// SIMATIC S7-200 project (STEP 7-Micro/WIN), CPU 224 CN REL 02.01

ORGANIZATION_BLOCK 主程序:OB1
TITLE=我们打算使用温度控制和数据监控确保水质处理效果。
// 具体的实现过程是这样的：系统通过模拟量输入通道接收温度传感器传来的0-20mA信号（对应0-32000的模拟值）。程序调用模拟量子程序，将信号转换为实际温度值，存储在工程值输出中。上限值设定为100.0°C，下限值设定为-50.0°C。当模拟量输入通道的值小于等于6400（对应4mA）时，工程值输出直接设为-50.0°C；当模拟量输入通道的值大于等于32000（对应20mA）时，工程值输出设为100.0°C；当模拟量输入通道的值在6400到32000之间时，通过线性插值计算出对应的温度，例如50.0°C。系统假设模拟量输入通道的值在0到32000之间，并且上限值设定大于下限值设定。
BEGIN
Network 1
LD     SM0.0
CALL   模拟量子程序:SBR3, AIW0, 100.0, -50.0, VD10
END_ORGANIZATION_BLOCK

// SBR1: protected block, not included

SUBROUTINE_BLOCK 模拟量子程序:SBR3
TITLE=
VAR_INPUT
AIW:INT;	// LW0 
HI:REAL;	// LD2 
LO:REAL;	// LD6 
END_VAR
VAR_OUTPUT
OUT:REAL;	// LD10 
END_VAR
BEGIN
Network 1 // 网络标题
// 0~20ma  对应0~32000
LD     SM0.0
ITD    #AIW:LW0, VD300
AENO
DTR    VD300, VD300
Network 2
LD     SM0.0
AR<=   VD300, 6400.0
MOVR   #LO:LD6, #OUT:LD10
Network 3
LD     SM0.0
AR>=   VD300, 32000.0
MOVR   #HI:LD2, #OUT:LD10
Network 4
LD     SM0.0
AR>    VD300, 6400.0
AR<    VD300, 32000.0
-R     6400.0, VD300
AENO
/R     25600.0, VD300
AENO
MOVR   VD300, #OUT:LD10
AENO
*R     VD304, #OUT:LD10
AENO
+R     #LO:LD6, #OUT:LD10
Network 5
LD     SM0.0
MOVR   #HI:LD2, VD304
-R     #LO:LD6, VD304
END_SUBROUTINE_BLOCK

// (further data pages could not be read)
